# EPICS substitutions: ek9000App/Db/EL1084.substitutions
file EL1084.template
{       pattern
        {
                TERMINAL,

        }
        {
        }
}
